PROGRAM pouAxis
VAR
	retvall: UDINT;
END_VAR

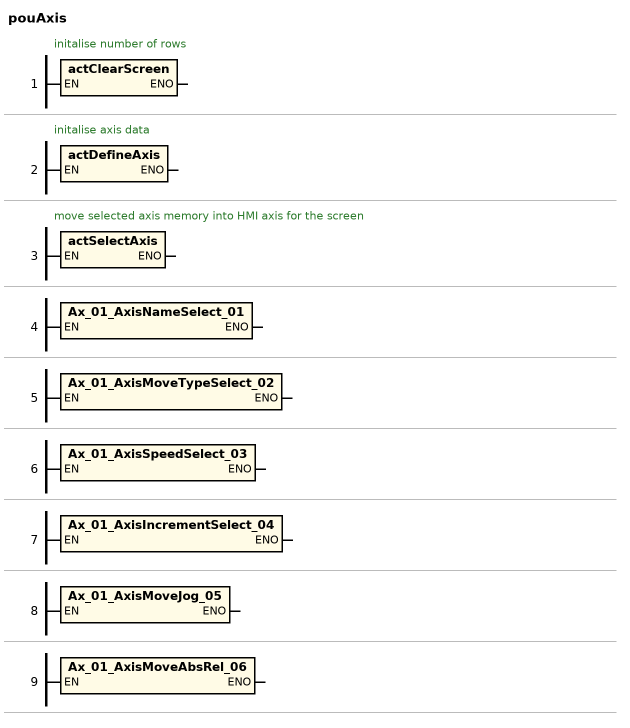
// NETWORK 1
// initalise number of rows
actClearScreen();

// NETWORK 2
// initalise axis data
actDefineAxis();

// NETWORK 3
// move selected axis memory into HMI axis for the screen
actSelectAxis();

// NETWORK 4
Ax_01_AxisNameSelect_01();

// NETWORK 5
Ax_01_AxisMoveTypeSelect_02();

// NETWORK 6
Ax_01_AxisSpeedSelect_03();

// NETWORK 7
Ax_01_AxisIncrementSelect_04();

// NETWORK 8
Ax_01_AxisMoveJog_05();

// NETWORK 9
Ax_01_AxisMoveAbsRel_06();

ACTION actClearScreen:
//clear HMI row for manual insertion
axis.gAxisRows.gMotionRow1.IndexLocation := 0;
axis.gAxisRows.gMotionRow2.IndexLocation := 20;
axis.gAxisRows.gMotionRow3.IndexLocation := 40;
axis.gAxisRows.gMotionRow4.IndexLocation := 60;
axis.gAxisRows.gMotionRow5.IndexLocation := 80;
axis.gAxisRows.gMotionRow6.IndexLocation := 100;

//clear axis row layout
axis.gAxisNumRows := 0;

//debug
axis.isAxisStandStill := TRUE;
END_ACTION

ACTION actDefineAxis:

//axis define for HMI screen feedback
Axis.axisPresent[1].AxisName := 'Gantry Traverse'; //name of axis
Axis.axisPresent[1].AxisDef := 'X'; //X,Y,Z, A,B,C, etc
Axis.axisPresent[1].AxisNumber := 1;
Axis.axisPresent[1].isLinearDrive := TRUE;
Axis.axisPresent[1].isSpindleDrive := FALSE;

//axis define for HMI screen feedback
Axis.axisPresent[2].AxisName := 'Gantry Raise/Lower'; //name of axis
Axis.axisPresent[2].AxisDef := 'Y'; //X,Y,Z, A,B,C, etc
Axis.axisPresent[2].AxisNumber := 2;
Axis.axisPresent[2].isLinearDrive := TRUE;
Axis.axisPresent[2].isSpindleDrive := FALSE;

//axis define for HMI screen feedback
Axis.axisPresent[3].AxisName := 'Gantry Clamp'; //name of axis
Axis.axisPresent[3].AxisDef := 'Z'; //X,Y,Z, A,B,C, etc
Axis.axisPresent[3].AxisNumber := 3;
Axis.axisPresent[3].isLinearDrive := TRUE;
Axis.axisPresent[3].isSpindleDrive := FALSE;

//axis define for HMI screen feedback
Axis.axisPresent[4].AxisName := 'Spindle 1'; //name of axis
Axis.axisPresent[4].AxisDef := 'S1'; //X,Y,Z, A,B,C, etc
Axis.axisPresent[4].AxisNumber := 4;
Axis.axisPresent[4].isLinearDrive := FALSE;
Axis.axisPresent[4].isSpindleDrive := TRUE;

//axis define for HMI screen feedback
Axis.axisPresent[5].AxisName := 'Spindle 2'; //name of axis
Axis.axisPresent[5].AxisDef := 'S2'; //X,Y,Z, A,B,C, etc
Axis.axisPresent[5].AxisNumber := 5;
Axis.axisPresent[5].isLinearDrive := FALSE;
Axis.axisPresent[5].isSpindleDrive := TRUE;

//axis define for HMI screen feedback
Axis.axisPresent[6].AxisName := 'Cleaning Brush'; //name of axis
Axis.axisPresent[6].AxisDef := 'A'; //X,Y,Z, A,B,C, etc
Axis.axisPresent[6].AxisNumber := 6;
Axis.axisPresent[6].isLinearDrive := TRUE;
Axis.axisPresent[6].isSpindleDrive := FALSE;

//define max axis useage
//could write a loop to work that out
Axis.gNumAxisInSystem := 6;
END_ACTION

ACTION actSelectAxis:
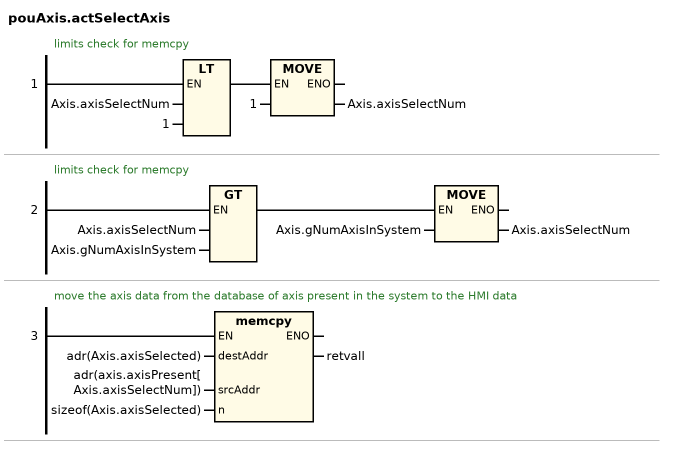
// NETWORK 1
// limits check for memcpy
IF Axis.axisSelectNum < 1 THEN Axis.axisSelectNum := 1; END_IF

// NETWORK 2
// limits check for memcpy
IF Axis.axisSelectNum > Axis.gNumAxisInSystem THEN Axis.axisSelectNum := Axis.gNumAxisInSystem; END_IF

// NETWORK 3
// move the axis data from the database of axis present in the system to the HMI data
retvall := memcpy(destAddr := adr(Axis.axisSelected), srcAddr := adr(axis.axisPresent[Axis.axisSelectNum]), n := sizeof(Axis.axisSelected));
END_ACTION

END_PROGRAM

(* stored: Version 1.1.0.1, ProductVersion 3.1.4024.12
   POU pouAxis: Id {0a1eb7e7-2ca7-4349-8d96-78253461d98b}, SpecialFunc None
   Action actClearScreen: Id {a9ff748a-de6a-4eb1-8d41-a39e8e6638f7}
   Action actDefineAxis: Id {9af7c28b-6d61-4a84-85ca-c2c5ea7f91d2}
   Action actSelectAxis: Id {e33c6345-de27-4668-8193-d15a263d3f2f} *)
